FUNCTION CheckDivDInt : DINT
VAR_INPUT
	divisor:DINT;
END_VAR

{noflow}
IF divisor = 0 THEN
	CheckDivDInt:=1;
	oaksGVL.udiCheckDivDInt := oaksGVL.udiCheckDivDInt + 1;
ELSE
	CheckDivDInt:=divisor;
END_IF;
{flow}

END_FUNCTION

(* stored: Version 1.1.0.1, ProductVersion 3.1.4022.18
   POU CheckDivDInt: Id {dfc0335d-9086-475f-8f1f-2e8877911b63}, SpecialFunc CheckDivInt32 *)
